// SIMATIC S7-200 project (STEP 7-Micro/WIN), CPU 224XP CN REL 02.01

ORGANIZATION_BLOCK MAIN:OB1
TITLE=PROGRAM COMMENTS
BEGIN
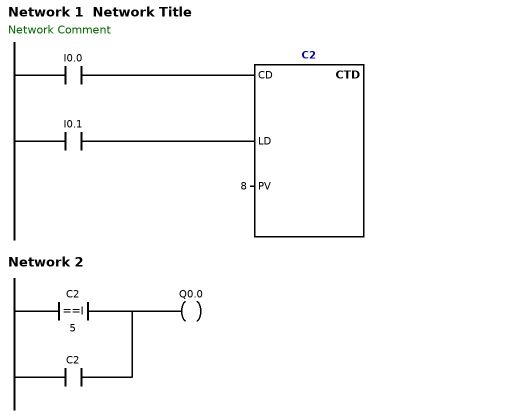
Network 1 // Network Title
// Network Comment
LD     I0.0
LD     I0.1
CTD    C2, 8
Network 2
LDW=   C2, 5
O      C2
=      Q0.0
END_ORGANIZATION_BLOCK
